SYSTEM Xplus3
  (* Version 1.0, Author, 4DIAC-Consortium *)
  APPLICATION Xplus3Application
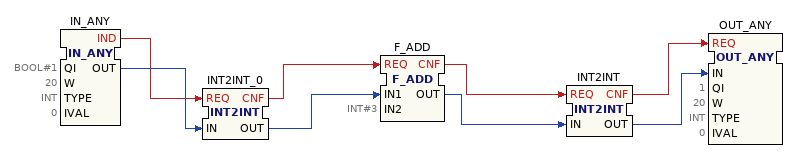
    FBS
      OUT_ANY : OUT_ANY(QI := 1, W := 20, TYPE := INT, IVAL := 0);
      INT2INT : INT2INT;
      INT2INT_0 : INT2INT;
      F_ADD : F_ADD(IN2 := INT#3);
      IN_ANY : IN_ANY(QI := BOOL#1, W := 20, TYPE := INT, IVAL := 0);
    END_FBS
    EVENT_CONNECTIONS
      INT2INT_0.CNF TO F_ADD.REQ;
      F_ADD.CNF TO INT2INT.REQ;
      IN_ANY.IND TO INT2INT_0.REQ;
      INT2INT.CNF TO OUT_ANY.REQ;
    END_CONNECTIONS
    DATA_CONNECTIONS
      INT2INT_0.OUT TO F_ADD.IN1;
      F_ADD.OUT TO INT2INT.IN;
      INT2INT.OUT TO OUT_ANY.IN;
      IN_ANY.OUT TO INT2INT_0.IN;
    END_CONNECTIONS
  END_APPLICATION
  DEVICE MICROCONTROLLER : FORTE_PC(MGR_ID := "localhost:61499")
    {SET_ATTRIBUTE(Profile, HOLOBLOC)}
    RESOURCE CALC : EMB_RES
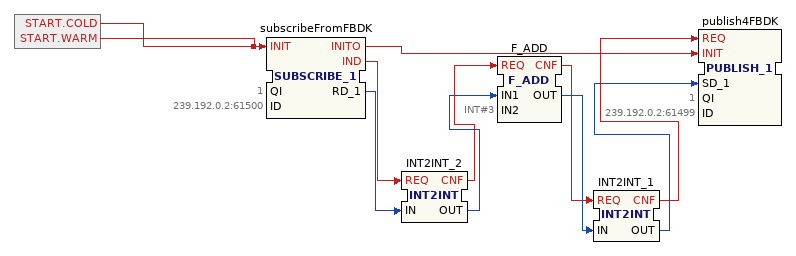
      FBS
        F_ADD : F_ADD(IN2 := INT#3);
        INT2INT_1 : INT2INT;
        INT2INT_2 : INT2INT;
        publish4FBDK : PUBLISH_1(QI := 1, ID := 239.192.0.2:61499);
        subscribeFromFBDK : SUBSCRIBE_1(QI := 1, ID := 239.192.0.2:61500);
      END_FBS
      EVENT_CONNECTIONS
        INT2INT_2.CNF TO F_ADD.REQ;
        F_ADD.CNF TO INT2INT_1.REQ;
        INT2INT_1.CNF TO publish4FBDK.REQ;
        subscribeFromFBDK.INITO TO publish4FBDK.INIT;
        START.COLD TO subscribeFromFBDK.INIT;
        START.WARM TO subscribeFromFBDK.INIT;
        subscribeFromFBDK.IND TO INT2INT_2.REQ;
      END_CONNECTIONS
      DATA_CONNECTIONS
        INT2INT_2.OUT TO F_ADD.IN1;
        F_ADD.OUT TO INT2INT_1.IN;
        INT2INT_1.OUT TO publish4FBDK.SD_1;
        subscribeFromFBDK.RD_1 TO INT2INT_2.IN;
      END_CONNECTIONS
    END_RESOURCE
  END_DEVICE
  DEVICE PC : FBRT_WINDOW(BOUNDS := [50,50,250,100], GRID := [1,1], MGR_ID := "localhost:61499")
    {SET_ATTRIBUTE(Profile, HOLOBLOC)}
    RESOURCE VIS : PANEL_RESOURCE
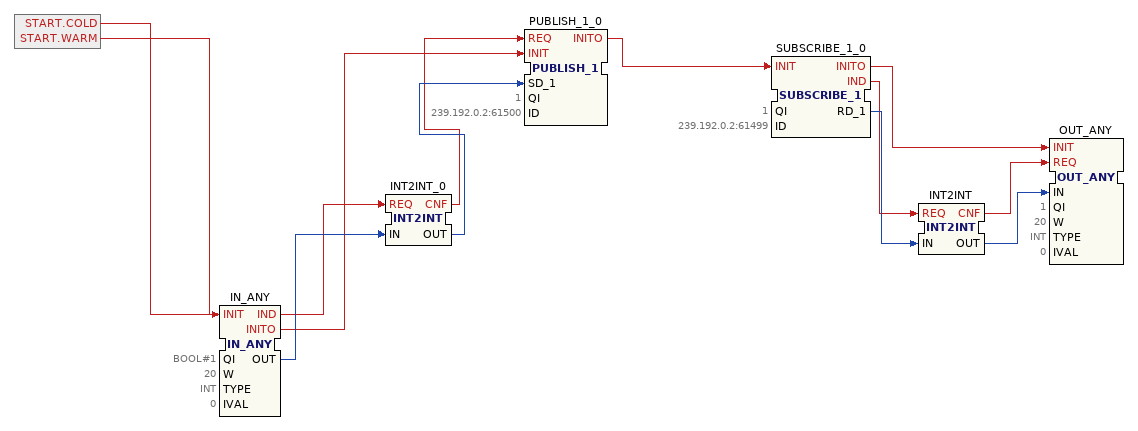
      FBS
        INT2INT_0 : INT2INT;
        INT2INT : INT2INT;
        OUT_ANY : OUT_ANY(QI := 1, W := 20, TYPE := INT, IVAL := 0);
        SUBSCRIBE_1_0 : SUBSCRIBE_1(QI := 1, ID := 239.192.0.2:61499);
        PUBLISH_1_0 : PUBLISH_1(QI := 1, ID := 239.192.0.2:61500);
        IN_ANY : IN_ANY(QI := BOOL#1, W := 20, TYPE := INT, IVAL := 0);
      END_FBS
      EVENT_CONNECTIONS
        PUBLISH_1_0.INITO TO SUBSCRIBE_1_0.INIT;
        SUBSCRIBE_1_0.INITO TO OUT_ANY.INIT;
        INT2INT_0.CNF TO PUBLISH_1_0.REQ;
        SUBSCRIBE_1_0.IND TO INT2INT.REQ;
        IN_ANY.IND TO INT2INT_0.REQ;
        START.COLD TO IN_ANY.INIT;
        START.WARM TO IN_ANY.INIT;
        IN_ANY.INITO TO PUBLISH_1_0.INIT;
        INT2INT.CNF TO OUT_ANY.REQ;
      END_CONNECTIONS
      DATA_CONNECTIONS
        INT2INT.OUT TO OUT_ANY.IN;
        INT2INT_0.OUT TO PUBLISH_1_0.SD_1;
        SUBSCRIBE_1_0.RD_1 TO INT2INT.IN;
        IN_ANY.OUT TO INT2INT_0.IN;
      END_CONNECTIONS
    END_RESOURCE
  END_DEVICE
  MAPPINGS
    Xplus3Application.OUT_ANY ON PC.VIS.OUT_ANY;
    Xplus3Application.INT2INT ON PC.VIS.INT2INT;
    Xplus3Application.INT2INT_0 ON PC.VIS.INT2INT_0;
    Xplus3Application.F_ADD ON MICROCONTROLLER.CALC.F_ADD;
    Xplus3Application.IN_ANY ON PC.VIS.IN_ANY;
  END_MAPPINGS
  SEGMENTS
    Ethernet : Ethernet;
  END_SEGMENTS
  LINKS
    MICROCONTROLLER => Ethernet;
    PC => Ethernet;
  END_LINKS
END_SYSTEM
